FUNCTION_BLOCK FLASHERW (* N-bit multimode Flasher *)
  (* Standard: 61499; Classification: Test; Function: Flasher; Type: 10 outputs *)
  (* Version 0.1, 2004-04-22, JHC, Rockwell Automation, Moved to fb.rt.math. *)
  (* Version 0.0, 2003-11-23, JHC, Rockwell Automation, Generalized from FLASHER10W. *)
  (* Compiler header: package fb.rt.math; *)
  (* Compiler Java Sun JDK 1.3.1 *)
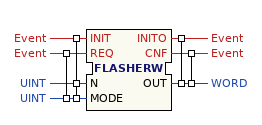
  EVENT_INPUT
    INIT WITH N, MODE; (* Initialization Request *)
    REQ WITH MODE; (* Update Request *)
  END_EVENT
  EVENT_OUTPUT
    INITO WITH OUT; (* Initialization Confirm *)
    CNF WITH OUT; (* Update Confirmation *)
  END_EVENT
  VAR_INPUT
    N : UINT := 16; (* Number of bits to flash (intenally limited to 0<N<17). *)
    MODE : UINT; (* 0=FLASH_ALL,1=COUNT_UP,2=COUNT_DOWN,3=CHASE_UP,4=CHASE_DOWN *)
  END_VAR
  VAR_OUTPUT
    OUT : WORD;
  END_VAR
END_FUNCTION_BLOCK
